// TIA Portal V21 export
FUNCTION_BLOCK "SyntheticCases_FB"   // FB0, LAD
{ S7_Optimized_Access := 'TRUE' }
// stored: SetENOAutomatically false
BEGIN

REGION Network 1
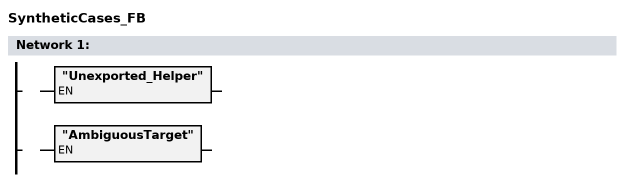
   "Unexported_Helper"();
   "AmbiguousTarget"();
END_REGION
END_FUNCTION_BLOCK
